{attribute 'enable_dynamic_creation'}
FUNCTION_BLOCK INTERNAL FB_SQLServerLogger IMPLEMENTS ILogger
VAR_INPUT
END_VAR
VAR_OUTPUT
END_VAR
VAR
END_VAR

METHOD PUBLIC Write : STRING
VAR_INPUT
	sMsg	: string;
END_VAR
Write := CONCAT('DatabaseLogger: ', sMsg);
END_METHOD

END_FUNCTION_BLOCK

(* stored: Version 1.1.0.1, ProductVersion 3.1.0.24
   POU FB_SQLServerLogger: Id {182f805a-1111-4214-be00-6e7a500a1623}
   Method Write: Id {cee6d0d4-852e-4ff4-b662-bbca5a63d315} *)
